INTERFACE IResult EXTENDS __SYSTEM.IQueryInterface

PROPERTY Busy : BOOL
GET
END_GET
SET
END_SET
END_PROPERTY

PROPERTY Done : BOOL
GET
END_GET
SET
END_SET
END_PROPERTY

PROPERTY Error : BOOL
GET
END_GET
SET
END_SET
END_PROPERTY

PROPERTY ErrorId : DINT
GET
END_GET
SET
END_SET
END_PROPERTY

END_INTERFACE

(* stored: Version 1.1.0.1, ProductVersion 3.1.4024.12
   Itf IResult: Id {a0b6e183-7d75-423f-8b8b-e47f2cd3f637}
   Property Busy: Id {1d74b76b-52bc-4cd2-a78f-2434322e2ff5}
   Get Get: Id {b49b738e-55f3-43cc-8424-45a3258cd540}
   Set Set: Id {45aa2dca-9572-432b-a4e7-73b1816695d2}
   Property Done: Id {9ea9d55d-8822-4de1-a02f-8cc1529a8a98}
   Get Get: Id {52acd90a-e8ce-4550-a38a-66b5352b02eb}
   Set Set: Id {ad59c078-b0ec-4267-9a84-0deaced04f83}
   Property Error: Id {9211bef2-0002-407a-b3be-5c87f20f68fd}
   Get Get: Id {63057b26-7677-4c6e-aa87-4bff642b88bb}
   Set Set: Id {f1b482f2-f993-4452-a09e-405377344913}
   Property ErrorId: Id {bef6ddca-305d-4a23-9e8b-1e1712f88a6d}
   Get Get: Id {9903dc13-a3ee-402c-aa91-b8eaeb5f04e2}
   Set Set: Id {a5cd992e-303a-4d76-8380-98f572defa56} *)
